
FUNCTION CB_mod_sint : INT


TITLE = ' Modulo of integer '
VERSION : '1.0'
AUTHOR  : CB
NAME    : modSint
FAMILY  : TNI

VAR_INPUT
    IN1 : INT;
    IN2 : INT;
END_VAR

BEGIN
    CB_mod_sint := IN1 MOD IN2;
END_FUNCTION
